FUNCTION_BLOCK Z_CONTROLLER2 (* HVAC Zone temperature panel controller *)
  (* Standard: 61499-2 *)
  (* Version 1.0, 2020-01-14, badger *)
  (* Compiler header: #include "Z_CONTROLLER_Library.cpp" *)
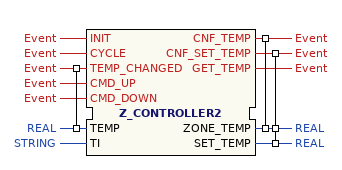
  EVENT_INPUT
    INIT; (* Initialises the zone controller *)
    CYCLE;
    TEMP_CHANGED WITH TEMP; (* The temperature in the zone has changed. *)
    CMD_UP; (* Signal that the zone set up switch has been pressed *)
    CMD_DOWN; (* Signal that the zone set down switch has been pressed *)
  END_EVENT
  EVENT_OUTPUT
    CNF_TEMP WITH ZONE_TEMP; (* Signals that the temperature in the zone has changed *)
    CNF_SET_TEMP WITH ZONE_TEMP, SET_TEMP; (* Signals that the set temperature in the zone has changed *)
    GET_TEMP; (* Request a new temperature reading *)
  END_EVENT
  VAR_INPUT
    TEMP : REAL; (* New temperature from the temperature probe *)
    TI : STRING;
  END_VAR
  VAR_OUTPUT
    ZONE_TEMP : REAL; (* Current temperature in the zone *)
    SET_TEMP : REAL; (* The set temperature in the zone *)
  END_VAR
  VAR
    ZONE_TEMPERATURE : REAL; (* Current zone temperature *)
    ZONE_SET_TEMPERATURE : REAL; (* Current zone set temperature *)
  END_VAR
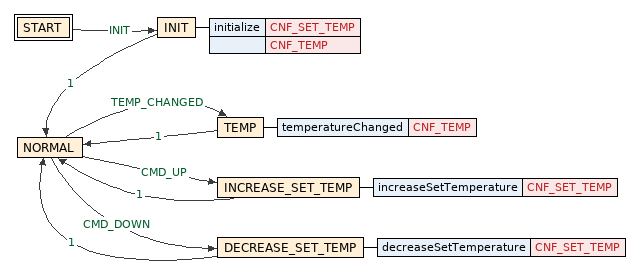
  EC_STATES
    START; (* Initial State *)
    INIT : initialize -> CNF_SET_TEMP, -> CNF_TEMP;
    NORMAL;
    TEMP : temperatureChanged -> CNF_TEMP;
    INCREASE_SET_TEMP : increaseSetTemperature -> CNF_SET_TEMP;
    DECREASE_SET_TEMP : decreaseSetTemperature -> CNF_SET_TEMP;
  END_STATES
  EC_TRANSITIONS
    START TO INIT := INIT;
    INIT TO NORMAL := 1;
    NORMAL TO TEMP := TEMP_CHANGED;
    TEMP TO NORMAL := 1;
    NORMAL TO INCREASE_SET_TEMP := CMD_UP;
    INCREASE_SET_TEMP TO NORMAL := 1;
    NORMAL TO DECREASE_SET_TEMP := CMD_DOWN;
    DECREASE_SET_TEMP TO NORMAL := 1;
  END_TRANSITIONS
  ALGORITHM initialize IN AnyText: (* Initialization algorithm *)
	cout << "[Z_CONTROLLER2] alg_initialize()\n";
	// Set default room temperature and zone temperature
	ZONE_TEMP() = 18.0;
	SET_TEMP() = 15.0;
  END_ALGORITHM
  ALGORITHM normalOperation IN AnyText: (* Normal quiesent operational state of the controller *)
	cout <<  "[Z_CONTROLLER2] alg_normalOperation\n";
  END_ALGORITHM
  ALGORITHM temperatureChanged IN AnyText: (* Zone temperature has changed *)
	cout << "[Z_CONTROLLER2] alg_temperatureChanged\n";
	ZONE_TEMP() = TEMP();
  END_ALGORITHM
  ALGORITHM increaseSetTemperature IN AnyText: (* Increase the set temperature by one degree *)
	cout << "[Z_CONTROLLER2] alg_increaseSetTemperature\n";
	SET_TEMP() = SET_TEMP() + 1.0;
  END_ALGORITHM
  ALGORITHM decreaseSetTemperature IN AnyText: (* Decrease the set temperature by one degree *)
	cout << "[Z_CONTROLLER2] alg_decreaseSetTemperature\n";
	SET_TEMP() = SET_TEMP() - 1.0;
  END_ALGORITHM
END_FUNCTION_BLOCK
